Staubli VAL3: calculate_pick.pgx

public program calculate_pick(num x_nNum_row, num x_nNum_col, point& x_pPoint_return, num x_nNum_choose)
  local num l_nNum_pitchX
  local num l_nNum_pitchY
  local point l_pPoint_lb
begin
  //given row,col(z-based, count from left-bottom)
  //return position


  //set left-bottom corner position and pitch
  switch x_nNum_choose
    case 1
      //f1
      l_nNum_pitchX = 6.6
      l_nNum_pitchY = 11.3

      l_pPoint_lb = pPointRx_f1_lb
    break
    case 2
      //f2
      l_nNum_pitchX = 8
      l_nNum_pitchY = 10

      l_pPoint_lb = pPointRx_f2_lb
    break
    case 3
      //f3
      l_nNum_pitchX = -14
      l_nNum_pitchY = 22

      l_pPoint_lb = pPointRx_f3_lb
    break
    case 4
      //bottom
      l_nNum_pitchX = 32
      l_nNum_pitchY = 33

      l_pPoint_lb = pPointRx_bt_lb
    break

  endSwitch


  x_pPoint_return = l_pPoint_lb

  x_pPoint_return.trsf.x = x_pPoint_return.trsf.x + x_nNum_col * l_nNum_pitchX
  x_pPoint_return.trsf.y = x_pPoint_return.trsf.y + x_nNum_row * l_nNum_pitchY

  //---------------------------------------------
  // Bottom part special case - base frame offset
  //---------------------------------------------
  switch x_nNum_choose
    case 4
      fFrame_ofs.trsf.x = x_nNum_col * l_nNum_pitchX
      fFrame_ofs.trsf.y = x_nNum_row * l_nNum_pitchY
      //maintain the lb point
      x_pPoint_return = pPointRx_bt_lb
    break
  endSwitch

end
